FUNCTION_BLOCK Leg_Control_Mapping_Model
VAR_INPUT
	Control_Leg		: ARRAY [1..18] OF LREAL;		// 控制程序中的腿编号
END_VAR
VAR_OUTPUT
	Model_Leg		: ARRAY [1..18] OF LREAL;		// 模型中的腿编号
END_VAR
VAR
END_VAR

Model_Leg[1]		:= Control_Leg[1];
Model_Leg[2]		:= Control_Leg[6];
Model_Leg[3]		:= Control_Leg[5];
Model_Leg[4]		:= Control_Leg[4];
Model_Leg[5]		:= Control_Leg[3];
Model_Leg[6]		:= Control_Leg[2];

END_FUNCTION_BLOCK

(* stored: Version 1.1.0.1, ProductVersion 3.1.4020.12
   POU Leg_Control_Mapping_Model: Id {061643dc-3529-42c6-8d6d-f250dae82188}, SpecialFunc None *)
